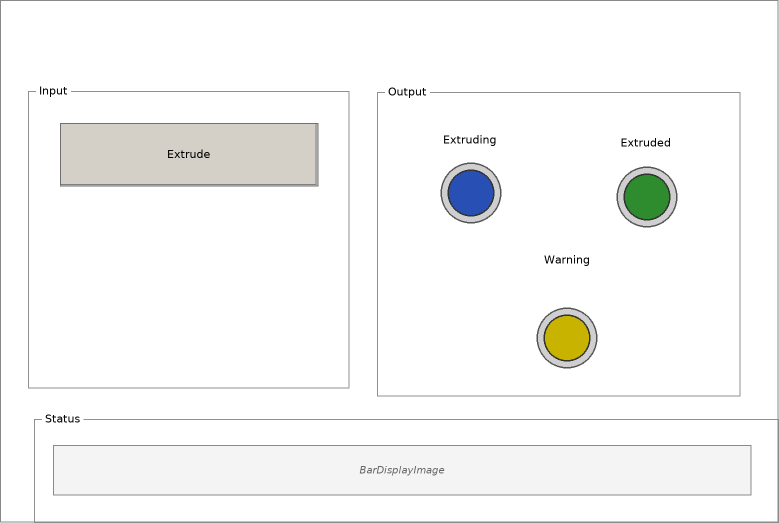
VISUALIZATION Visualization  // 779x523
    GroupBox (28,83 321x305), "Input"
        Button (32,40 258x63), "Extrude"
            OnMouseClick: execute { Q10.extrude := TRUE; }
    GroupBox (377,84 363x312), "Output"
        Lamp1 (59,74 70x70), variable: Q10.extruding, style: Lamp-Lamp1-Blue
        Lamp1 (155,219 70x70), variable: Q10.warning, style: Lamp-Lamp1-Yellow
        Label (18,41 150x30), "Extruding"
        Label (194,44 150x30), "Extruded"
        Label (115,161 150x30), "Warning"
        Lamp1 (235,78 70x70), variable: Q10.extruded, style: Lamp-Lamp1-Green
    GroupBox (34,411 745x112), "Status"
        BarDisplayImage (19,34 698x50), value: Q10.count_i, style: BarDisplayImage-Gray, scale format: %.1f, scale 0..20000
END_VISUALIZATION

(* stored: Version 1.1.0.1, ProductVersion 3.1.4024.12
   Visu Visualization: Id {3c6b89e6-c123-4c5b-8a48-18c0e1800d3e} *)
